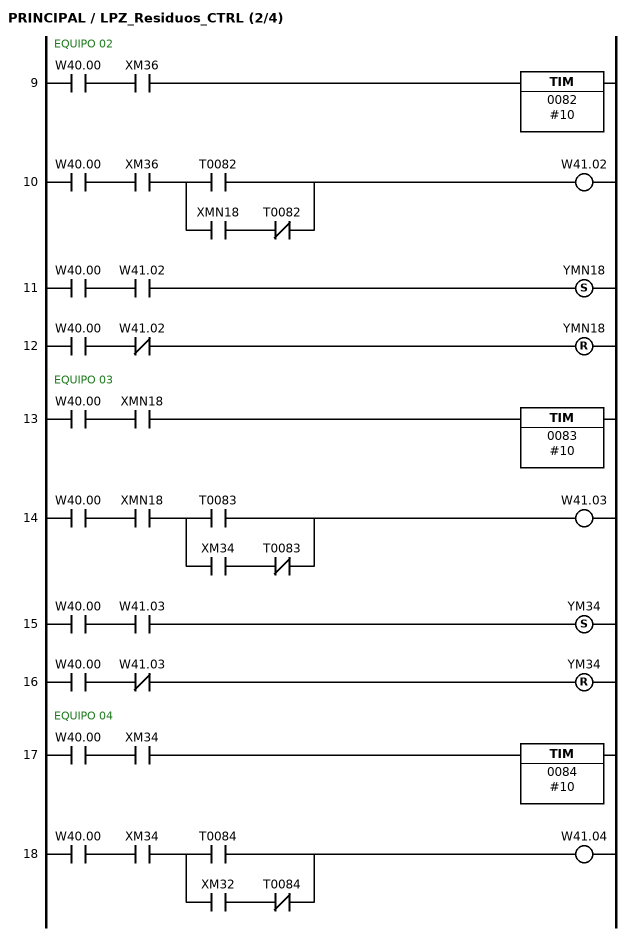
; [picture p48: PRINCIPAL / LPZ_Residuos_CTRL, rungs 9-18]
; rung 9: EQUIPO 02
LD W40.00
AND XM36
TIM 0082 #10
; rung 10
LD W40.00
AND XM36
LD T0082
LD XMN18
ANDNOT T0082
ORLD
ANDLD
OUT W41.02
; rung 11
LD W40.00
AND W41.02
SET YMN18
; rung 12
LD W40.00
ANDNOT W41.02
RSET YMN18
; rung 13: EQUIPO 03
LD W40.00
AND XMN18
TIM 0083 #10
; rung 14
LD W40.00
AND XMN18
LD T0083
LD XM34
ANDNOT T0083
ORLD
ANDLD
OUT W41.03
; rung 15
LD W40.00
AND W41.03
SET YM34
; rung 16
LD W40.00
ANDNOT W41.03
RSET YM34
; rung 17: EQUIPO 04
LD W40.00
AND XM34
TIM 0084 #10
; rung 18
LD W40.00
AND XM34
LD T0084
LD XM32
ANDNOT T0084
ORLD
ANDLD
OUT W41.04

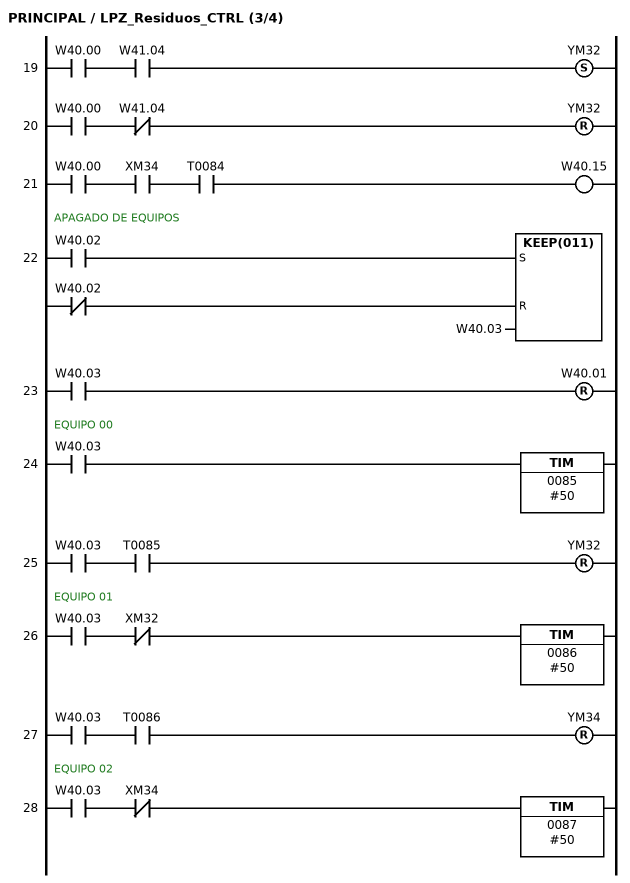
; rung 19
LD W40.00
AND W41.04
SET YM32
; rung 20
LD W40.00
ANDNOT W41.04
RSET YM32
; rung 21
LD W40.00
AND XM34
AND T0084
OUT W40.15
; rung 22: APAGADO DE EQUIPOS
LD W40.02
LDNOT W40.02
KEEP(011) W40.03
; rung 23
LD W40.03
RSET W40.01
; rung 24: EQUIPO 00
LD W40.03
TIM 0085 #50
; rung 25
LD W40.03
AND T0085
RSET YM32
; rung 26: EQUIPO 01
LD W40.03
ANDNOT XM32
TIM 0086 #50
; rung 27
LD W40.03
AND T0086
RSET YM34
; rung 28: EQUIPO 02
LD W40.03
ANDNOT XM34
TIM 0087 #50

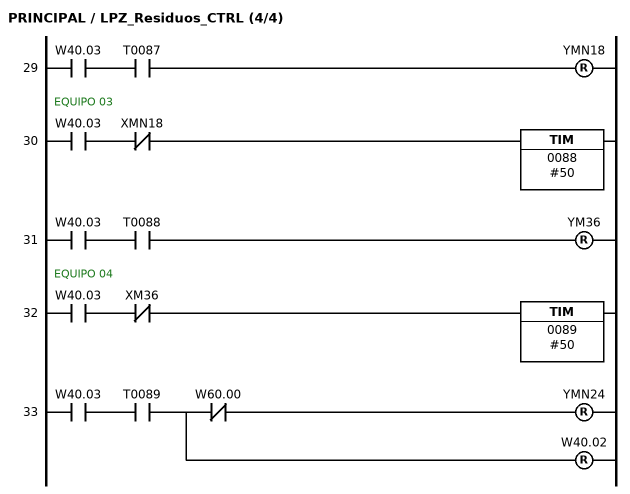
; rung 29
LD W40.03
AND T0087
RSET YMN18
; rung 30: EQUIPO 03
LD W40.03
ANDNOT XMN18
TIM 0088 #50
; rung 31
LD W40.03
AND T0088
RSET YM36
; rung 32: EQUIPO 04
LD W40.03
ANDNOT XM36
TIM 0089 #50
; rung 33
LD W40.03
AND T0089
OUT TR0
ANDNOT W60.00
RSET YMN24
LD TR0
RSET W40.02

### Section LPZ_Residuos_OUT

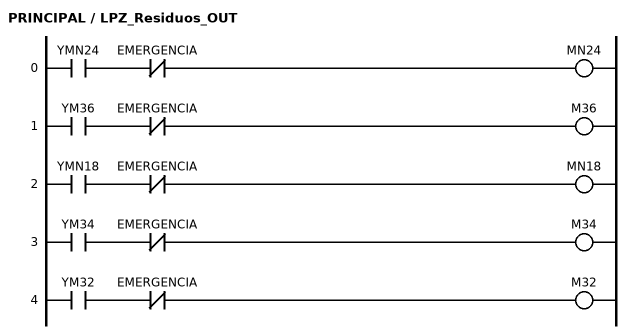
; rung 0
LD YMN24
ANDNOT EMERGENCIA
OUT MN24
; rung 1
LD YM36
ANDNOT EMERGENCIA
OUT M36
; rung 2
LD YMN18
ANDNOT EMERGENCIA
OUT MN18
; rung 3
LD YM34
ANDNOT EMERGENCIA
OUT M34
; rung 4
LD YM32
ANDNOT EMERGENCIA
OUT M32

### Section LPZ_Ventilador_CTRL

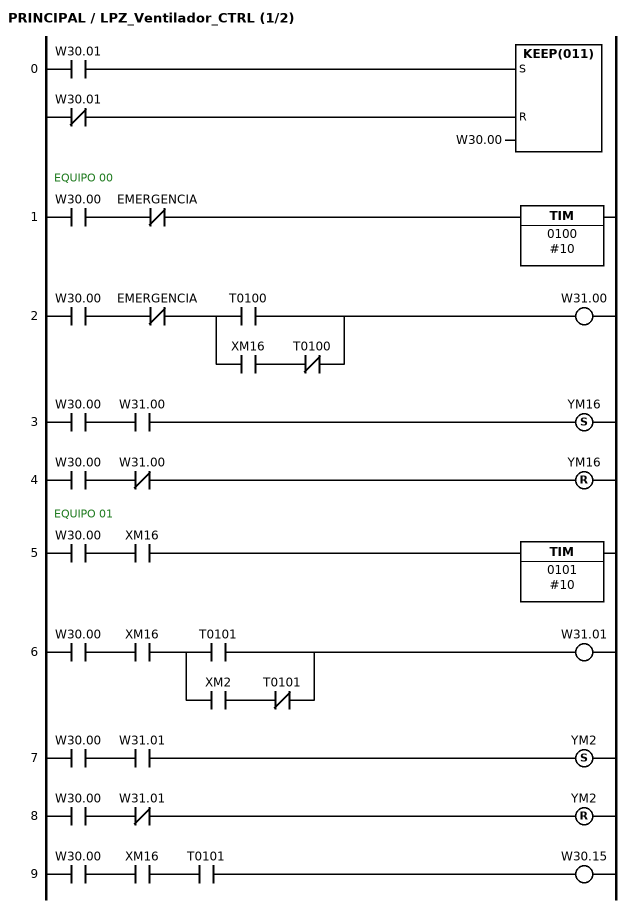
; rung 0
LD W30.01
LDNOT W30.01
KEEP(011) W30.00
; rung 1: EQUIPO 00
LD W30.00
ANDNOT EMERGENCIA
TIM 0100 #10
; rung 2
LD W30.00
ANDNOT EMERGENCIA
LD T0100
LD XM16
ANDNOT T0100
ORLD
ANDLD
OUT W31.00
; rung 3
LD W30.00
AND W31.00
SET YM16
; rung 4
LD W30.00
ANDNOT W31.00
RSET YM16
; rung 5: EQUIPO 01
LD W30.00
AND XM16
TIM 0101 #10
; rung 6
LD W30.00
AND XM16
LD T0101
LD XM2
ANDNOT T0101
ORLD
ANDLD
OUT W31.01
; rung 7
LD W30.00
AND W31.01
SET YM2
; rung 8
LD W30.00
ANDNOT W31.01
RSET YM2
; rung 9
LD W30.00
AND XM16
AND T0101
OUT W30.15

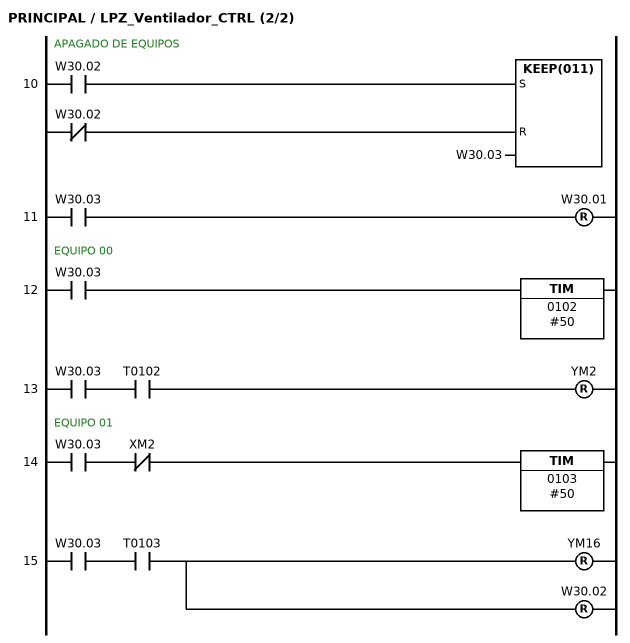
; rung 10: APAGADO DE EQUIPOS
LD W30.02
LDNOT W30.02
KEEP(011) W30.03
; rung 11
LD W30.03
RSET W30.01
; rung 12: EQUIPO 00
LD W30.03
TIM 0102 #50
; rung 13
LD W30.03
AND T0102
RSET YM2
; rung 14: EQUIPO 01
LD W30.03
ANDNOT XM2
TIM 0103 #50
; rung 15
LD W30.03
AND T0103
RSET YM16
RSET W30.02

### Section LPZ_Ventilador_OUT

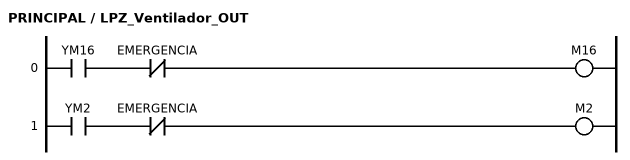
; rung 0
LD YM16
ANDNOT EMERGENCIA
OUT M16
; rung 1
LD YM2
ANDNOT EMERGENCIA
OUT M2

### Section LPZ_1Rociado_CTRL

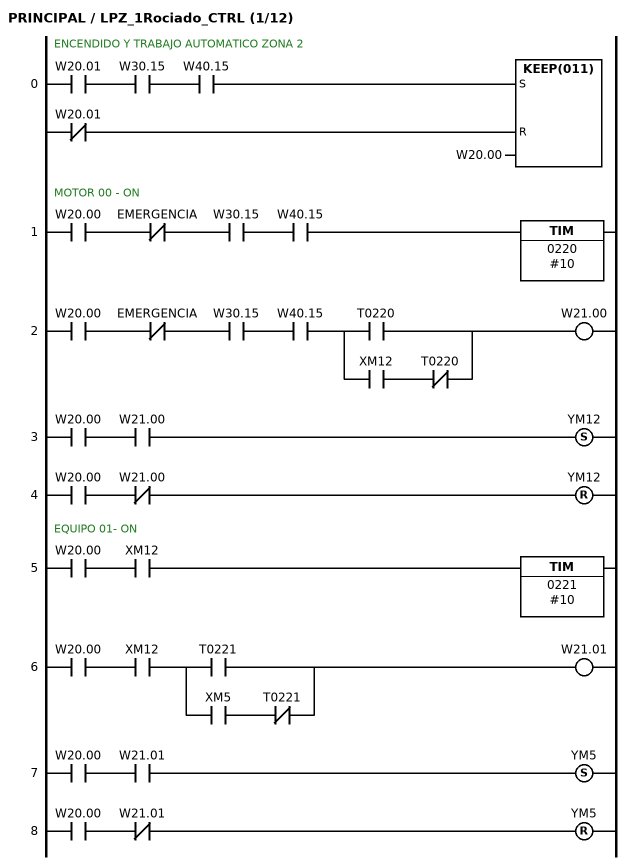
; rung 0: ENCENDIDO Y TRABAJO AUTOMATICO ZONA 2
LD W20.01
AND W30.15
AND W40.15
LDNOT W20.01
KEEP(011) W20.00
; rung 1: MOTOR 00 - ON
LD W20.00
ANDNOT EMERGENCIA
AND W30.15
AND W40.15
TIM 0220 #10
; rung 2
LD W20.00
ANDNOT EMERGENCIA
AND W30.15
AND W40.15
LD T0220
LD XM12
ANDNOT T0220
ORLD
ANDLD
OUT W21.00
; rung 3
LD W20.00
AND W21.00
SET YM12
; rung 4
LD W20.00
ANDNOT W21.00
RSET YM12
; rung 5: EQUIPO 01- ON
LD W20.00
AND XM12
TIM 0221 #10
; rung 6
LD W20.00
AND XM12
LD T0221
LD XM5
ANDNOT T0221
ORLD
ANDLD
OUT W21.01
; rung 7
LD W20.00
AND W21.01
SET YM5
; rung 8
LD W20.00
ANDNOT W21.01
RSET YM5

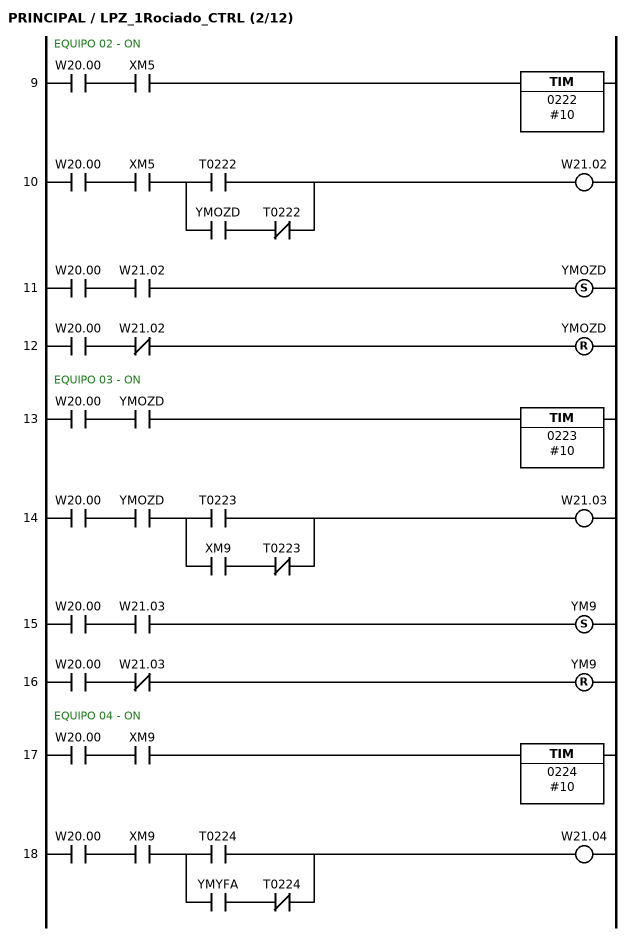
; rung 9: EQUIPO 02 - ON
LD W20.00
AND XM5
TIM 0222 #10
; rung 10
LD W20.00
AND XM5
LD T0222
LD YMOZD
ANDNOT T0222
ORLD
ANDLD
OUT W21.02
; rung 11
LD W20.00
AND W21.02
SET YMOZD
; rung 12
LD W20.00
ANDNOT W21.02
RSET YMOZD
; rung 13: EQUIPO 03 - ON
LD W20.00
AND YMOZD
TIM 0223 #10
; rung 14
LD W20.00
AND YMOZD
LD T0223
LD XM9
ANDNOT T0223
ORLD
ANDLD
OUT W21.03
; rung 15
LD W20.00
AND W21.03
SET YM9
; rung 16
LD W20.00
ANDNOT W21.03
RSET YM9
; rung 17: EQUIPO 04 - ON
LD W20.00
AND XM9
TIM 0224 #10
; rung 18
LD W20.00
AND XM9
LD T0224
LD YMYFA
ANDNOT T0224
ORLD
ANDLD
OUT W21.04

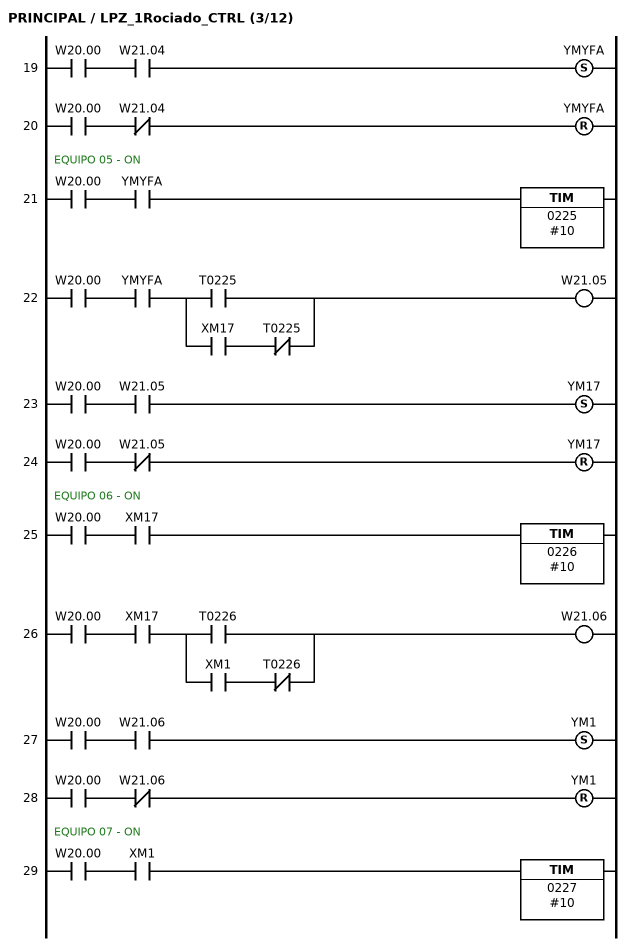
; rung 19
LD W20.00
AND W21.04
SET YMYFA
; rung 20
LD W20.00
ANDNOT W21.04
RSET YMYFA
; rung 21: EQUIPO 05 - ON
LD W20.00
AND YMYFA
TIM 0225 #10
; rung 22
LD W20.00
AND YMYFA
LD T0225
LD XM17
ANDNOT T0225
ORLD
ANDLD
OUT W21.05
; rung 23
LD W20.00
AND W21.05
SET YM17
; rung 24
LD W20.00
ANDNOT W21.05
RSET YM17
; rung 25: EQUIPO 06 - ON
LD W20.00
AND XM17
TIM 0226 #10
; rung 26
LD W20.00
AND XM17
LD T0226
LD XM1
ANDNOT T0226
ORLD
ANDLD
OUT W21.06
; rung 27
LD W20.00
AND W21.06
SET YM1
; rung 28
LD W20.00
ANDNOT W21.06
RSET YM1
; rung 29: EQUIPO 07 - ON
LD W20.00
AND XM1
TIM 0227 #10

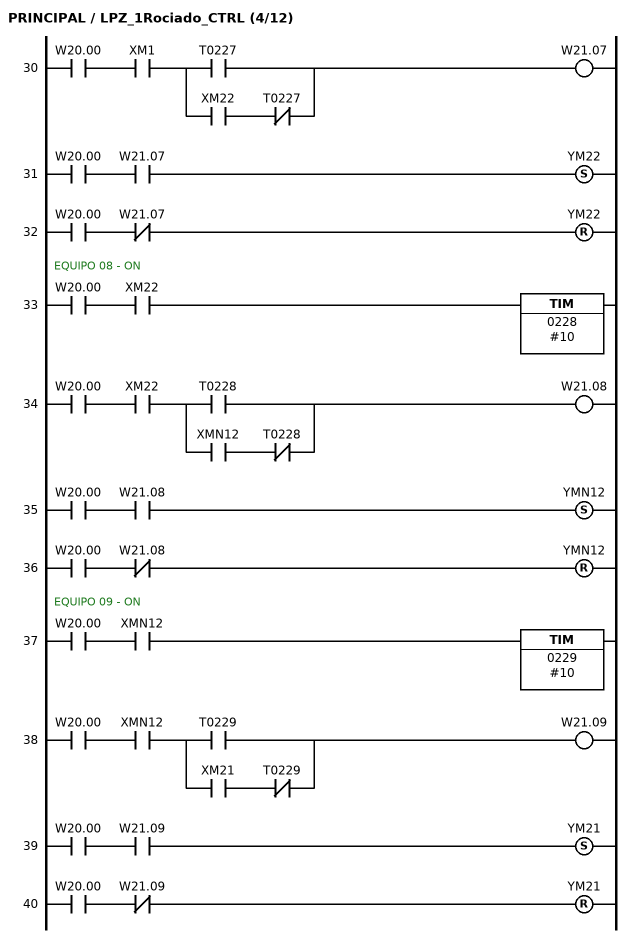
; rung 30
LD W20.00
AND XM1
LD T0227
LD XM22
ANDNOT T0227
ORLD
ANDLD
OUT W21.07
; rung 31
LD W20.00
AND W21.07
SET YM22
; rung 32
LD W20.00
ANDNOT W21.07
RSET YM22
; rung 33: EQUIPO 08 - ON
LD W20.00
AND XM22
TIM 0228 #10
; rung 34
LD W20.00
AND XM22
LD T0228
LD XMN12
ANDNOT T0228
ORLD
ANDLD
OUT W21.08
; rung 35
LD W20.00
AND W21.08
SET YMN12
; rung 36
LD W20.00
ANDNOT W21.08
RSET YMN12
; rung 37: EQUIPO 09 - ON
LD W20.00
AND XMN12
TIM 0229 #10
; rung 38
LD W20.00
AND XMN12
LD T0229
LD XM21
ANDNOT T0229
ORLD
ANDLD
OUT W21.09
; rung 39
LD W20.00
AND W21.09
SET YM21
; rung 40
LD W20.00
ANDNOT W21.09
RSET YM21

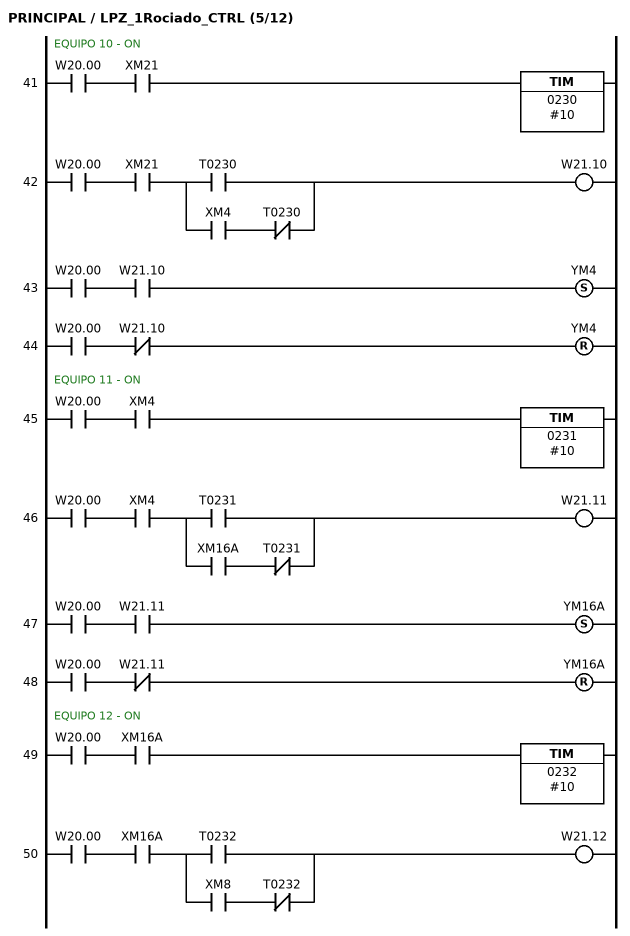
; rung 41: EQUIPO 10 - ON
LD W20.00
AND XM21
TIM 0230 #10
; rung 42
LD W20.00
AND XM21
LD T0230
LD XM4
ANDNOT T0230
ORLD
ANDLD
OUT W21.10
; rung 43
LD W20.00
AND W21.10
SET YM4
; rung 44
LD W20.00
ANDNOT W21.10
RSET YM4
; rung 45: EQUIPO 11 - ON
LD W20.00
AND XM4
TIM 0231 #10
; rung 46
LD W20.00
AND XM4
LD T0231
LD XM16A
ANDNOT T0231
ORLD
ANDLD
OUT W21.11
; rung 47
LD W20.00
AND W21.11
SET YM16A
; rung 48
LD W20.00
ANDNOT W21.11
RSET YM16A
; rung 49: EQUIPO 12 - ON
LD W20.00
AND XM16A
TIM 0232 #10
; rung 50
LD W20.00
AND XM16A
LD T0232
LD XM8
ANDNOT T0232
ORLD
ANDLD
OUT W21.12

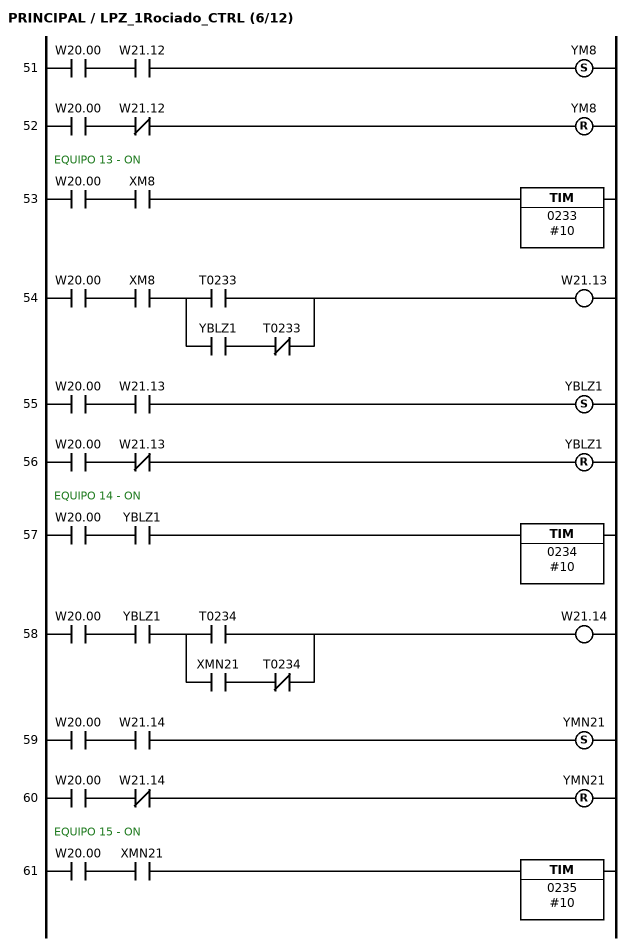
; rung 51
LD W20.00
AND W21.12
SET YM8
; rung 52
LD W20.00
ANDNOT W21.12
RSET YM8
; rung 53: EQUIPO 13 - ON
LD W20.00
AND XM8
TIM 0233 #10
; rung 54
LD W20.00
AND XM8
LD T0233
LD YBLZ1
ANDNOT T0233
ORLD
ANDLD
OUT W21.13
; rung 55
LD W20.00
AND W21.13
SET YBLZ1
; rung 56
LD W20.00
ANDNOT W21.13
RSET YBLZ1
; rung 57: EQUIPO 14 - ON
LD W20.00
AND YBLZ1
TIM 0234 #10
; rung 58
LD W20.00
AND YBLZ1
LD T0234
LD XMN21
ANDNOT T0234
ORLD
ANDLD
OUT W21.14
; rung 59
LD W20.00
AND W21.14
SET YMN21
; rung 60
LD W20.00
ANDNOT W21.14
RSET YMN21
; rung 61: EQUIPO 15 - ON
LD W20.00
AND XMN21
TIM 0235 #10

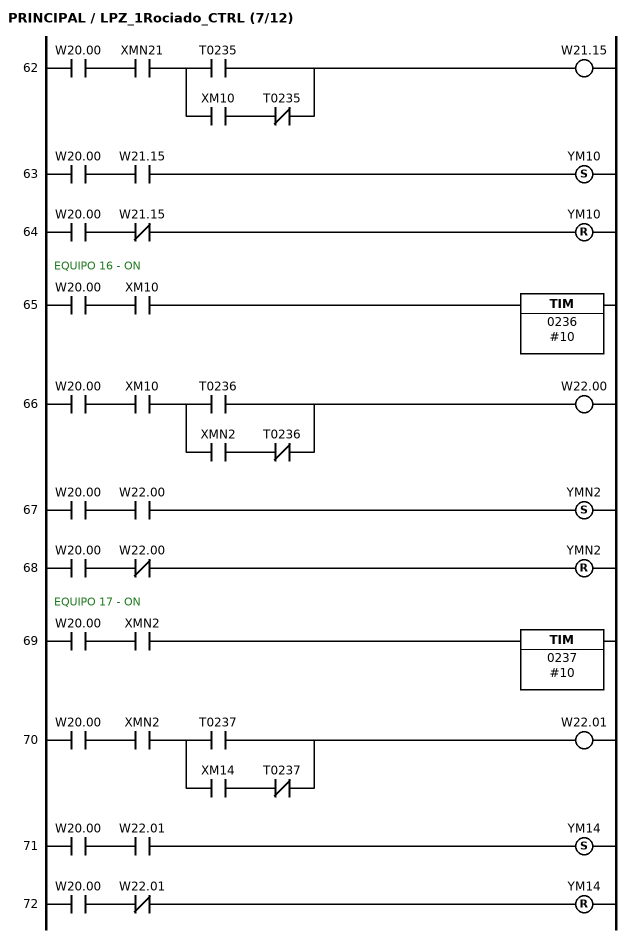
; rung 62
LD W20.00
AND XMN21
LD T0235
LD XM10
ANDNOT T0235
ORLD
ANDLD
OUT W21.15
; rung 63
LD W20.00
AND W21.15
SET YM10
; rung 64
LD W20.00
ANDNOT W21.15
RSET YM10
; rung 65: EQUIPO 16 - ON
LD W20.00
AND XM10
TIM 0236 #10
; rung 66
LD W20.00
AND XM10
LD T0236
LD XMN2
ANDNOT T0236
ORLD
ANDLD
OUT W22.00
; rung 67
LD W20.00
AND W22.00
SET YMN2
; rung 68
LD W20.00
ANDNOT W22.00
RSET YMN2
; rung 69: EQUIPO 17 - ON
LD W20.00
AND XMN2
TIM 0237 #10
; rung 70
LD W20.00
AND XMN2
LD T0237
LD XM14
ANDNOT T0237
ORLD
ANDLD
OUT W22.01
; rung 71
LD W20.00
AND W22.01
SET YM14
; rung 72
LD W20.00
ANDNOT W22.01
RSET YM14

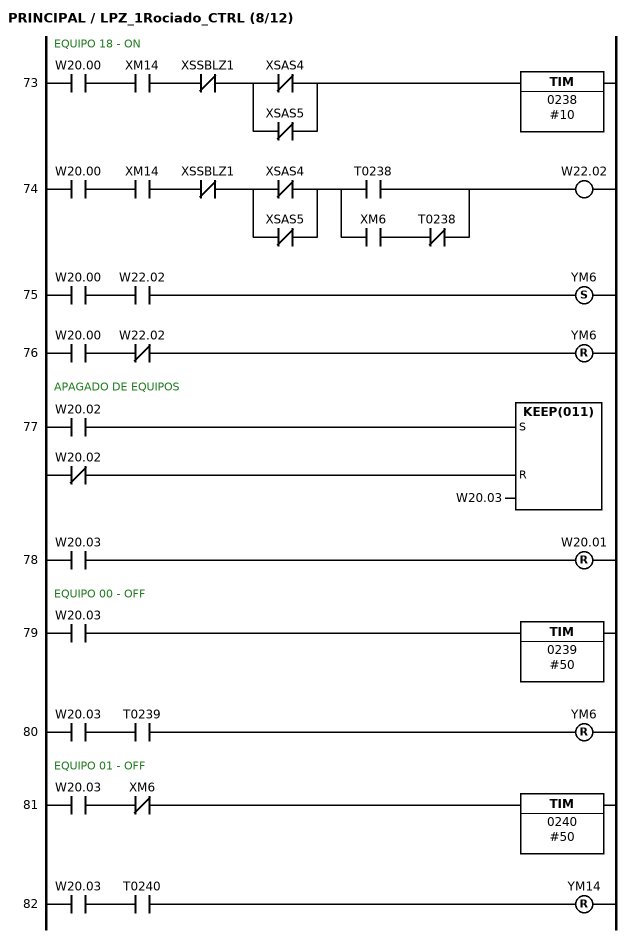
; rung 73: EQUIPO 18 - ON
LD W20.00
AND XM14
ANDNOT XSSBLZ1
LDNOT XSAS4
ORNOT XSAS5
ANDLD
TIM 0238 #10
; rung 74
LD W20.00
AND XM14
ANDNOT XSSBLZ1
LDNOT XSAS4
ORNOT XSAS5
ANDLD
LD T0238
LD XM6
ANDNOT T0238
ORLD
ANDLD
OUT W22.02
; rung 75
LD W20.00
AND W22.02
SET YM6
; rung 76
LD W20.00
ANDNOT W22.02
RSET YM6
; rung 77: APAGADO DE EQUIPOS
LD W20.02
LDNOT W20.02
KEEP(011) W20.03
; rung 78
LD W20.03
RSET W20.01
; rung 79: EQUIPO 00 - OFF
LD W20.03
TIM 0239 #50
; rung 80
LD W20.03
AND T0239
RSET YM6
; rung 81: EQUIPO 01 - OFF
LD W20.03
ANDNOT XM6
TIM 0240 #50
; rung 82
LD W20.03
AND T0240
RSET YM14

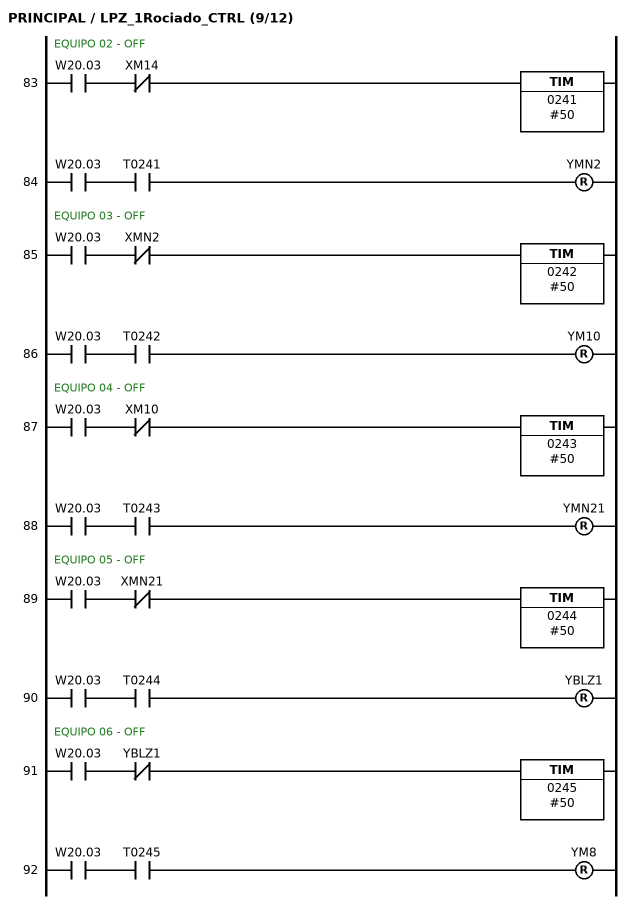
; rung 83: EQUIPO 02 - OFF
LD W20.03
ANDNOT XM14
TIM 0241 #50
; rung 84
LD W20.03
AND T0241
RSET YMN2
; rung 85: EQUIPO 03 - OFF
LD W20.03
ANDNOT XMN2
TIM 0242 #50
; rung 86
LD W20.03
AND T0242
RSET YM10
; rung 87: EQUIPO 04 - OFF
LD W20.03
ANDNOT XM10
TIM 0243 #50
; rung 88
LD W20.03
AND T0243
RSET YMN21
; rung 89: EQUIPO 05 - OFF
LD W20.03
ANDNOT XMN21
TIM 0244 #50
; rung 90
LD W20.03
AND T0244
RSET YBLZ1
; rung 91: EQUIPO 06 - OFF
LD W20.03
ANDNOT YBLZ1
TIM 0245 #50
; rung 92
LD W20.03
AND T0245
RSET YM8

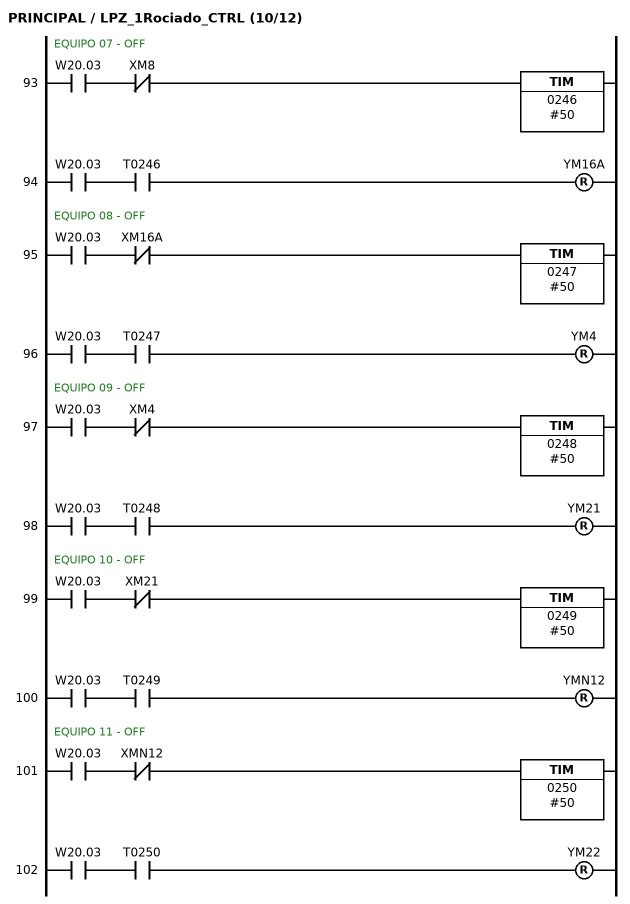
; rung 93: EQUIPO 07 - OFF
LD W20.03
ANDNOT XM8
TIM 0246 #50
; rung 94
LD W20.03
AND T0246
RSET YM16A
; rung 95: EQUIPO 08 - OFF
LD W20.03
ANDNOT XM16A
TIM 0247 #50
; rung 96
LD W20.03
AND T0247
RSET YM4
; rung 97: EQUIPO 09 - OFF
LD W20.03
ANDNOT XM4
TIM 0248 #50
; rung 98
LD W20.03
AND T0248
RSET YM21
; rung 99: EQUIPO 10 - OFF
LD W20.03
ANDNOT XM21
TIM 0249 #50
; rung 100
LD W20.03
AND T0249
RSET YMN12
; rung 101: EQUIPO 11 - OFF
LD W20.03
ANDNOT XMN12
TIM 0250 #50
; rung 102
LD W20.03
AND T0250
RSET YM22

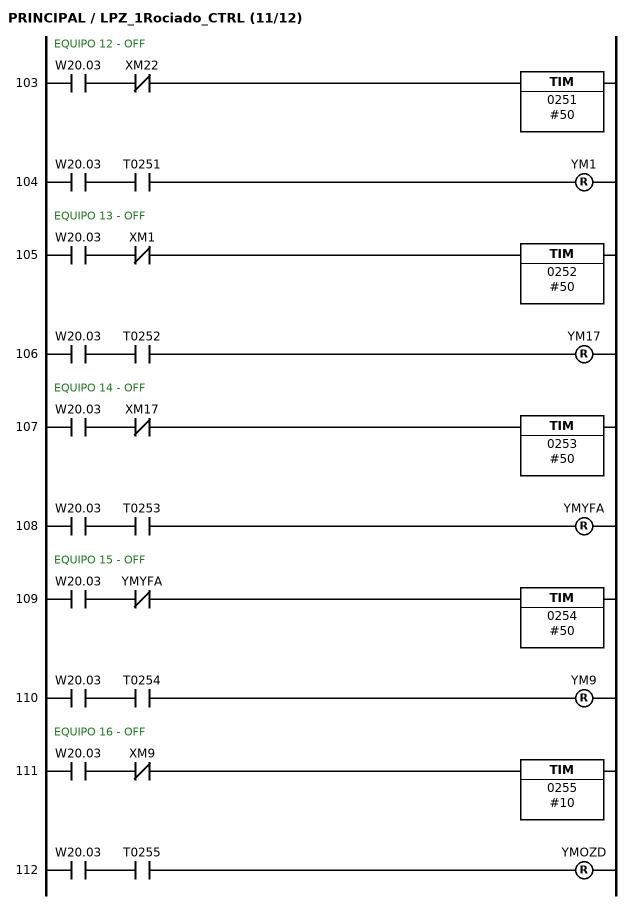
; rung 103: EQUIPO 12 - OFF
LD W20.03
ANDNOT XM22
TIM 0251 #50
; rung 104
LD W20.03
AND T0251
RSET YM1
; rung 105: EQUIPO 13 - OFF
LD W20.03
ANDNOT XM1
TIM 0252 #50
; rung 106
LD W20.03
AND T0252
RSET YM17
; rung 107: EQUIPO 14 - OFF
LD W20.03
ANDNOT XM17
TIM 0253 #50
; rung 108
LD W20.03
AND T0253
RSET YMYFA
; rung 109: EQUIPO 15 - OFF
LD W20.03
ANDNOT YMYFA
TIM 0254 #50
; rung 110
LD W20.03
AND T0254
RSET YM9
; rung 111: EQUIPO 16 - OFF
LD W20.03
ANDNOT XM9
TIM 0255 #10
; rung 112
LD W20.03
AND T0255
RSET YMOZD

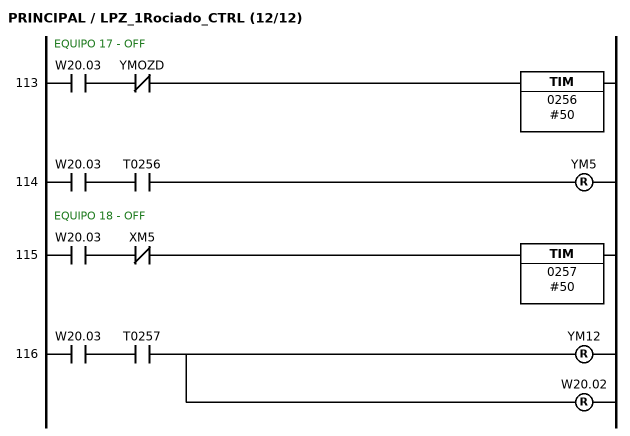
; rung 113: EQUIPO 17 - OFF
LD W20.03
ANDNOT YMOZD
TIM 0256 #50
; rung 114
LD W20.03
AND T0256
RSET YM5
; rung 115: EQUIPO 18 - OFF
LD W20.03
ANDNOT XM5
TIM 0257 #50
; rung 116
LD W20.03
AND T0257
RSET YM12
RSET W20.02

### Section LPZ_1Rociado_OUT

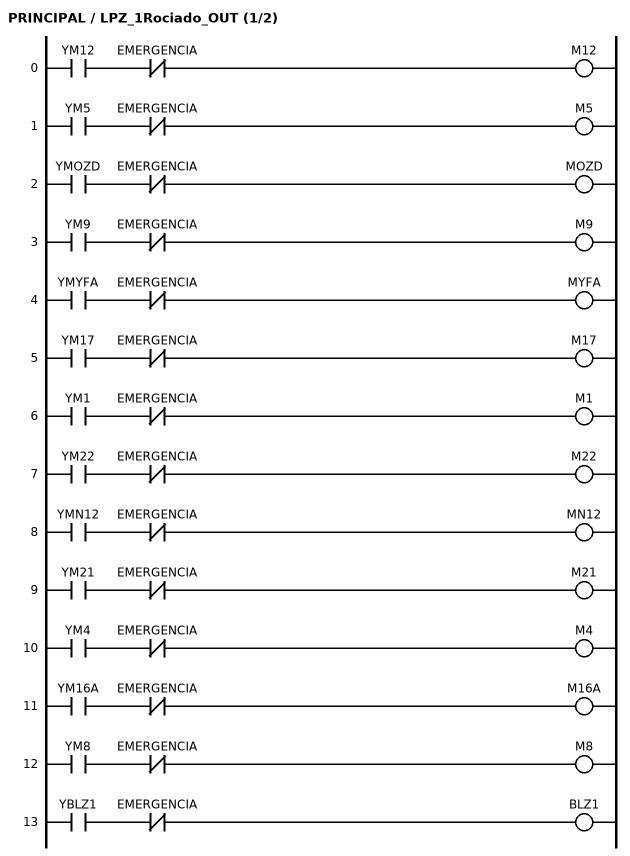
; rung 0
LD YM12
ANDNOT EMERGENCIA
OUT M12
; rung 1
LD YM5
ANDNOT EMERGENCIA
OUT M5
; rung 2
LD YMOZD
ANDNOT EMERGENCIA
OUT MOZD
; rung 3
LD YM9
ANDNOT EMERGENCIA
OUT M9
; rung 4
LD YMYFA
ANDNOT EMERGENCIA
OUT MYFA
; rung 5
LD YM17
ANDNOT EMERGENCIA
OUT M17
; rung 6
LD YM1
ANDNOT EMERGENCIA
OUT M1
; rung 7
LD YM22
ANDNOT EMERGENCIA
OUT M22
; rung 8
LD YMN12
ANDNOT EMERGENCIA
OUT MN12
; rung 9
LD YM21
ANDNOT EMERGENCIA
OUT M21
; rung 10
LD YM4
ANDNOT EMERGENCIA
OUT M4
; rung 11
LD YM16A
ANDNOT EMERGENCIA
OUT M16A
; rung 12
LD YM8
ANDNOT EMERGENCIA
OUT M8
; rung 13
LD YBLZ1
ANDNOT EMERGENCIA
OUT BLZ1

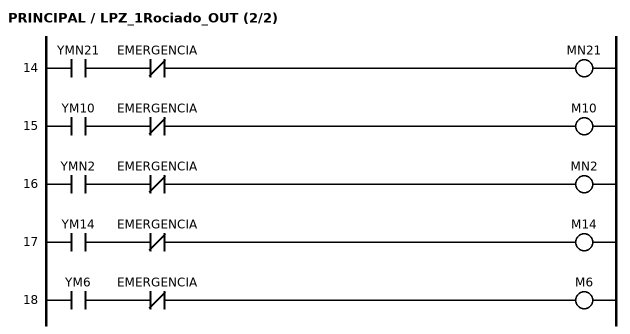
; rung 14
LD YMN21
ANDNOT EMERGENCIA
OUT MN21
; rung 15
LD YM10
ANDNOT EMERGENCIA
OUT M10
; rung 16
LD YMN2
ANDNOT EMERGENCIA
OUT MN2
; rung 17
LD YM14
ANDNOT EMERGENCIA
OUT M14
; rung 18
LD YM6
ANDNOT EMERGENCIA
OUT M6

### Section Molienda_OUT

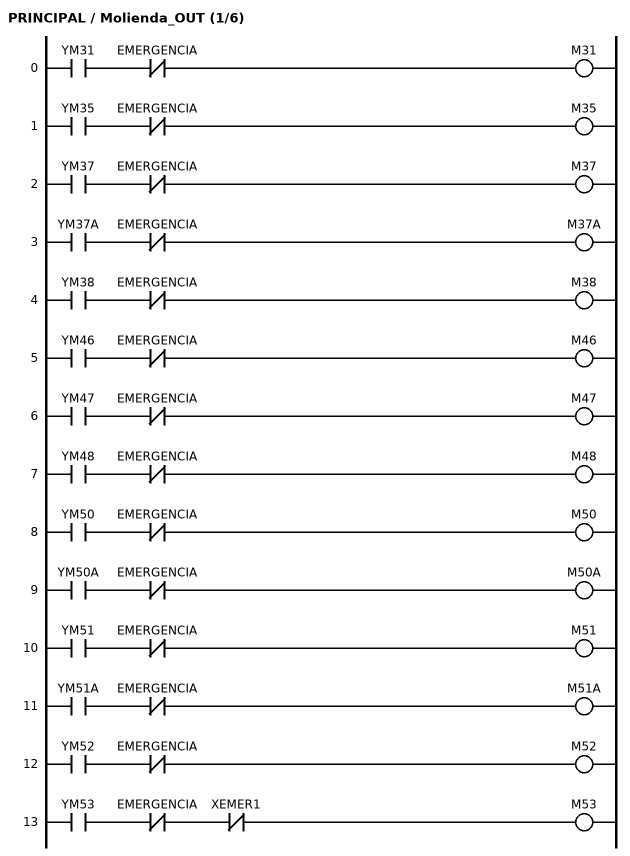
; rung 0
LD YM31
ANDNOT EMERGENCIA
OUT M31
; rung 1
LD YM35
ANDNOT EMERGENCIA
OUT M35
; rung 2
LD YM37
ANDNOT EMERGENCIA
OUT M37
; rung 3
LD YM37A
ANDNOT EMERGENCIA
OUT M37A
; rung 4
LD YM38
ANDNOT EMERGENCIA
OUT M38
; rung 5
LD YM46
ANDNOT EMERGENCIA
OUT M46
; rung 6
LD YM47
ANDNOT EMERGENCIA
OUT M47
; rung 7
LD YM48
ANDNOT EMERGENCIA
OUT M48
; rung 8
LD YM50
ANDNOT EMERGENCIA
OUT M50
; rung 9
LD YM50A
ANDNOT EMERGENCIA
OUT M50A
; rung 10
LD YM51
ANDNOT EMERGENCIA
OUT M51
; rung 11
LD YM51A
ANDNOT EMERGENCIA
OUT M51A
; rung 12
LD YM52
ANDNOT EMERGENCIA
OUT M52
; rung 13
LD YM53
ANDNOT EMERGENCIA
ANDNOT XEMER1
OUT M53

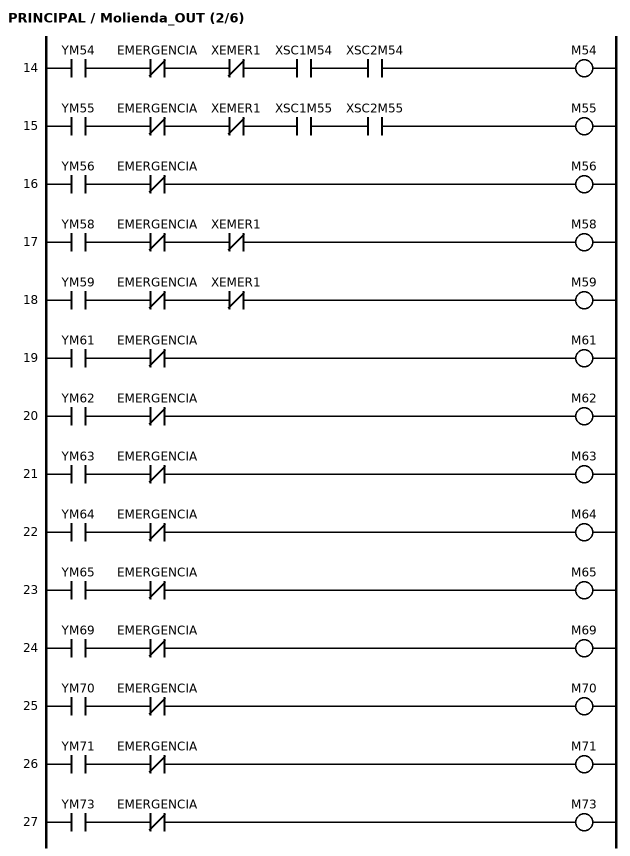
; rung 14
LD YM54
ANDNOT EMERGENCIA
ANDNOT XEMER1
AND XSC1M54
AND XSC2M54
OUT M54
; rung 15
LD YM55
ANDNOT EMERGENCIA
ANDNOT XEMER1
AND XSC1M55
AND XSC2M55
OUT M55
; rung 16
LD YM56
ANDNOT EMERGENCIA
OUT M56
; rung 17
LD YM58
ANDNOT EMERGENCIA
ANDNOT XEMER1
OUT M58
; rung 18
LD YM59
ANDNOT EMERGENCIA
ANDNOT XEMER1
OUT M59
; rung 19
LD YM61
ANDNOT EMERGENCIA
OUT M61
; rung 20
LD YM62
ANDNOT EMERGENCIA
OUT M62
; rung 21
LD YM63
ANDNOT EMERGENCIA
OUT M63
; rung 22
LD YM64
ANDNOT EMERGENCIA
OUT M64
; rung 23
LD YM65
ANDNOT EMERGENCIA
OUT M65
; rung 24
LD YM69
ANDNOT EMERGENCIA
OUT M69
; rung 25
LD YM70
ANDNOT EMERGENCIA
OUT M70
; rung 26
LD YM71
ANDNOT EMERGENCIA
OUT M71
; rung 27
LD YM73
ANDNOT EMERGENCIA
OUT M73

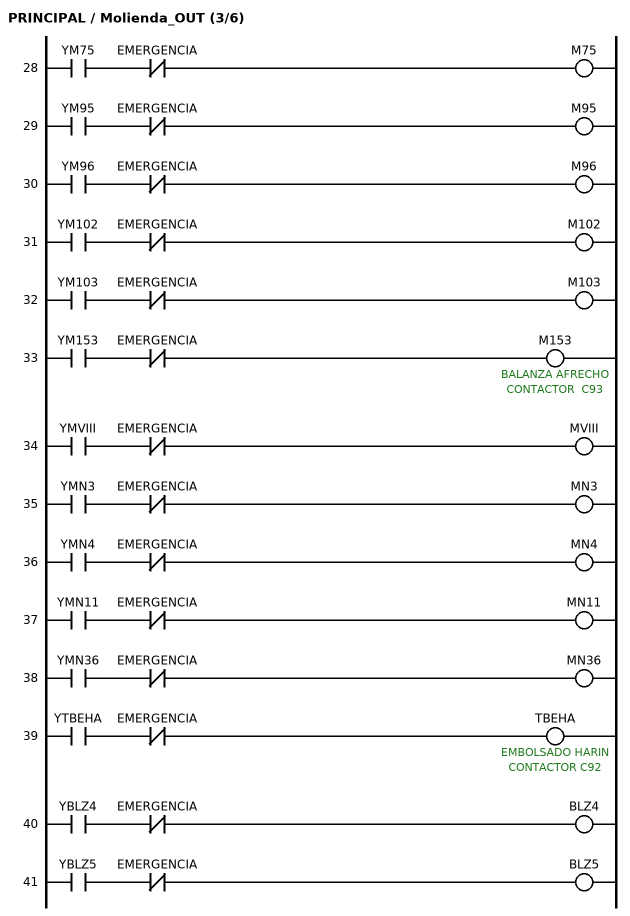
; rung 28
LD YM75
ANDNOT EMERGENCIA
OUT M75
; rung 29
LD YM95
ANDNOT EMERGENCIA
OUT M95
; rung 30
LD YM96
ANDNOT EMERGENCIA
OUT M96
; rung 31
LD YM102
ANDNOT EMERGENCIA
OUT M102
; rung 32
LD YM103
ANDNOT EMERGENCIA
OUT M103
; rung 33
LD YM153
ANDNOT EMERGENCIA
OUT M153  ; BALANZA AFRECHO CONTACTOR  C93
; rung 34
LD YMVIII
ANDNOT EMERGENCIA
OUT MVIII
; rung 35
LD YMN3
ANDNOT EMERGENCIA
OUT MN3
; rung 36
LD YMN4
ANDNOT EMERGENCIA
OUT MN4
; rung 37
LD YMN11
ANDNOT EMERGENCIA
OUT MN11
; rung 38
LD YMN36
ANDNOT EMERGENCIA
OUT MN36
; rung 39
LD YTBEHA
ANDNOT EMERGENCIA
OUT TBEHA  ; EMBOLSADO HARIN CONTACTOR C92
; rung 40
LD YBLZ4
ANDNOT EMERGENCIA
OUT BLZ4
; rung 41
LD YBLZ5
ANDNOT EMERGENCIA
OUT BLZ5

